{attribute 'GeneratedUsingTerminal: AX8108-0100-0101-0101'}
{attribute addProperty BoxType "AX8108-0100-0101-0101"}
{attribute addProperty Id "Ch_A_Target_positionAT %Q*DINT4Ch_A_Target_velocityAT %Q*DINT4"}
{attribute addProperty CRC "1177181981"}
{attribute addProperty Size "8"}
TYPE Ch_A_Interpolator_Outputs_462A5F1D :
STRUCT
	{attribute addProperty Name "Ch_A_Target_position"}
	Ch_A_Target_position AT %Q* : DINT;
	{attribute addProperty Name "Ch_A_Target_velocity"}
	Ch_A_Target_velocity AT %Q* : DINT;
END_STRUCT
END_TYPE
